{attribute 'Tc2GvlVarNames'}
VAR_CONFIG
END_VAR

(* stored: Version 1.1.0.1, ProductVersion 3.1.4024.9
   GVL Variable_Configuration: Id {9d0af4d4-35f8-4fce-8588-536927accf9e} *)
